// SIMATIC S7-200 SMART project (STEP 7-Micro/WIN SMART), CPU SR40

ORGANIZATION_BLOCK 主程序:OB1
TITLE=
BEGIN
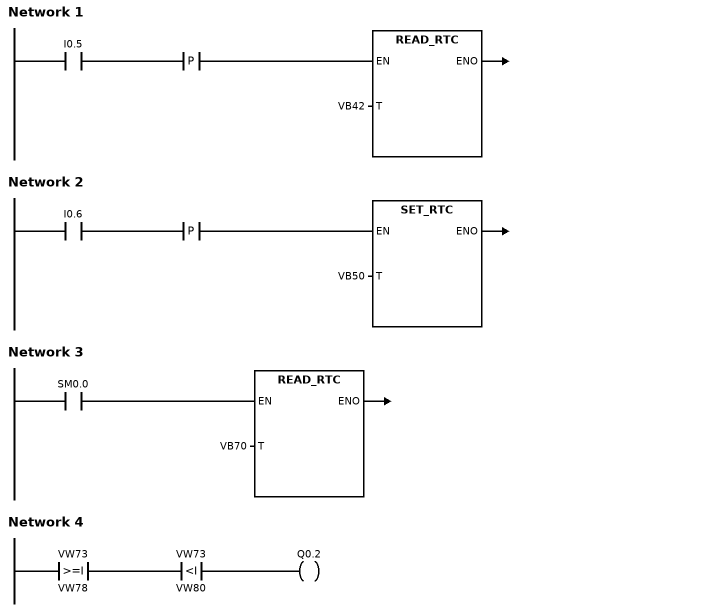
Network 1
LD     I0.5
EU
TODR   VB42
Network 2
LD     I0.6
EU
TODW   VB50
Network 3
LD     SM0.0
TODR   VB70
Network 4
LDW>=  VW73, VW78
AW<    VW73, VW80
=      Q0.2
END_ORGANIZATION_BLOCK
